PROGRAM Check_Filter
VAR
	Change_Filter : BOOL;
END_VAR

IF GVL_AirKnife.AirKnife_Start THEN
	IF GVL_AirKnife.AirKnife_Filter_Change_Setting <= GVL_AirKnife.AirKnife_Vacuum_Level THEN
		Change_Filter := TRUE;
	END_IF
ELSE
		Change_Filter := FALSE;
END_IF

END_PROGRAM

(* stored: Version 1.1.0.1, ProductVersion 3.1.4024.12
   POU Check_Filter: Id {523ae28a-dfdb-4838-a9ab-aefc8dd43478}, SpecialFunc None *)
